# B&R Automation Studio project EFI (part 11)

#### StackMethods.st
```iecst
ACTION StackMethods:

	IF NOT dataHeigh.status.xNewMediaStackEnabled THEN
		EnteringMediaContinuous.Media := dataHeigh.parameters.ContinuousMedia.MediaData;
	END_IF

	ReviewLoadNewMediaMethod;
	ReviewInsertNewMedia;
	ReviewRemoveNewMedia;

	ReviewLoadNewMediaEnergyMethod;
	ReviewInsertNewMediaEnMethod;

	ReviewLoadNewMediaEnergyContMethod;

	dataHeigh.status.Stack.iNewMediaLoadedL1 := Stack_iTotalNewMediaL1;
	dataHeigh.status.Stack.iNewMediaLoadedL2 := Stack_iTotalNewMediaL2;

END_ACTION

ACTION ReviewLoadNewMediaMethod:

	CASE LoadNewMedia_Step OF
		0: // Manage errors and init
			LoadNewMedia_Step := 1;

		1: // start operate
			LoadNewMedia_MethodOperate.Action  := UaMoa_CheckIsCalled;
			LoadNewMedia_MethodOperate.MethodName := 'LoadNewMedia';
			LoadNewMedia_MethodOperate.Execute := TRUE;
			LoadNewMedia_Step := 2;
		2: // check if method called
			LoadNewMedia_MethodOperate();
			IF LoadNewMedia_MethodOperate.Busy THEN
				LoadNewMedia_MethodOperate.Execute := FALSE;
			ELSE
				IF LoadNewMedia_MethodOperate.Done THEN
					LoadNewMedia_ErrorID:= 0;
					IF LoadNewMedia_MethodOperate.IsCalled THEN
						LoadNewMedia_Step := 3; // method is called
					END_IF
					LoadNewMedia_MethodOperate.Execute := TRUE;
				END_IF
				IF LoadNewMedia_MethodOperate.Error THEN
					LoadNewMedia_ErrorID:= DWORD_TO_UDINT(LoadNewMedia_MethodOperate.ErrorID);
					LoadNewMedia_Step := 0;
				END_IF
			END_IF
		3: // execute method code and return value
			ExecuteLoadingNewMedia;
			LoadNewMedia_Result := LoadNewMedia_ReviewResult;
			LoadNewMedia_Step := 4;
		4: // finish operate

			LoadNewMedia_MethodOperate.Action  := UaMoa_Finished;
			LoadNewMedia_MethodOperate.MethodName := 'LoadNewMedia';
			LoadNewMedia_MethodOperate.Execute := TRUE;
			LoadNewMedia_Step := 5;
		5: // finish method
			LoadNewMedia_MethodOperate();
			IF LoadNewMedia_MethodOperate.Busy THEN
				LoadNewMedia_MethodOperate.Execute := FALSE;
			ELSE
				IF LoadNewMedia_MethodOperate.Done THEN
					LoadNewMedia_ErrorID:= 0;
					LoadNewMedia_Step := 1; // method is finished, wait again for call
				END_IF
				IF LoadNewMedia_MethodOperate.Error THEN
					LoadNewMedia_ErrorID:= DWORD_TO_UDINT(LoadNewMedia_MethodOperate.ErrorID);
					LoadNewMedia_Step := 0;
				END_IF
			END_IF
	END_CASE

END_ACTION

ACTION ExecuteLoadingNewMedia:

	LoadNewMedia_ReviewResult := CheckMediaToStack(LoadNewMedia_Media,
												dataHeigh.status.xNewMediaStackEnabled,
												dataHeigh.parameters.xDoubleLine,
												25,
												200, 1400,
												200, 3000,
												Stack_iTotalNewMediaL1 >= THICK_MEDIATRACKING_MAX_MEDIA,
												Stack_iTotalNewMediaL2 >= THICK_MEDIATRACKING_MAX_MEDIA);

	IF LoadNewMedia_ReviewResult <> 0 THEN
		RETURN;
	END_IF

	// TODO: Load the media in the FIFO to manage it
	IF LoadNewMedia_Media.iLine = 1 THEN
		LoadNewMedia_ReviewResult := AssignLastItemInStack(
			ADR(LoadNewMedia_Media),
			ADR(NewMediaStackL1),
			Stack_iTotalNewMediaL1);

	ELSIF LoadNewMedia_Media.iLine = 2 THEN
		LoadNewMedia_ReviewResult := AssignLastItemInStack(
			ADR(LoadNewMedia_Media),
			ADR(NewMediaStackL2),
			Stack_iTotalNewMediaL2);

	END_IF

END_ACTION

ACTION ReviewInsertNewMedia:

	CASE InsertNewMedia_Step OF
		0: // Manage errors and init
			InsertNewMedia_Step := 1;

		1: // start operate
			InsertNewMedia_MethodOperate.Action  := UaMoa_CheckIsCalled;
			InsertNewMedia_MethodOperate.MethodName := 'InsertNewMedia';
			InsertNewMedia_MethodOperate.Execute := TRUE;
			InsertNewMedia_Step := 2;
		2: // check if method called
			InsertNewMedia_MethodOperate();
			IF InsertNewMedia_MethodOperate.Busy THEN
				InsertNewMedia_MethodOperate.Execute := FALSE;
			ELSE
				IF InsertNewMedia_MethodOperate.Done THEN
					InsertNewMedia_ErrorID:= 0;
					IF InsertNewMedia_MethodOperate.IsCalled THEN
						InsertNewMedia_Step := 3; // method is called
					END_IF
					InsertNewMedia_MethodOperate.Execute := TRUE;
				END_IF
				IF InsertNewMedia_MethodOperate.Error THEN
					InsertNewMedia_ErrorID:= DWORD_TO_UDINT(InsertNewMedia_MethodOperate.ErrorID);
					InsertNewMedia_Step := 0;
				END_IF
			END_IF
		3: // execute method code and return value
			ExecuteInsertNewMedia;
			InsertNewMedia_Result := InsertNewMedia_ReviewResult;
			InsertNewMedia_Step := 4;
		4: // finish operate

			InsertNewMedia_MethodOperate.Action  := UaMoa_Finished;
			InsertNewMedia_MethodOperate.MethodName := 'InsertNewMedia';
			InsertNewMedia_MethodOperate.Execute := TRUE;
			InsertNewMedia_Step := 5;
		5: // finish method
			InsertNewMedia_MethodOperate();
			IF InsertNewMedia_MethodOperate.Busy THEN
				InsertNewMedia_MethodOperate.Execute := FALSE;
			ELSE
				IF InsertNewMedia_MethodOperate.Done THEN
					InsertNewMedia_ErrorID:= 0;
					InsertNewMedia_Step := 1; // method is finished, wait again for call
				END_IF
				IF InsertNewMedia_MethodOperate.Error THEN
					InsertNewMedia_ErrorID:= DWORD_TO_UDINT(InsertNewMedia_MethodOperate.ErrorID);
					InsertNewMedia_Step := 0;
				END_IF
			END_IF
	END_CASE

END_ACTION

ACTION ExecuteInsertNewMedia:

	InsertNewMedia_ReviewResult := CheckMediaToStack(InsertNewMedia_Media,
												dataHeigh.status.xNewMediaStackEnabled,
												dataHeigh.parameters.xDoubleLine,
												25,
												200, 1400,
												200, 3000,
												Stack_iTotalNewMediaL1 >= THICK_MEDIATRACKING_MAX_MEDIA,
												Stack_iTotalNewMediaL2 >= THICK_MEDIATRACKING_MAX_MEDIA);

	IF InsertNewMedia_ReviewResult <> 0 THEN
		RETURN;
	END_IF

	// Load the media in the FIFO to manage it.
	// If an error occurs, the error is stored to return it in the method
	IF InsertNewMedia_Media.iLine = 1 THEN
		InsertNewMedia_ReviewResult := InsertItemInStack(
			InsertNewMedia_Id,
			ADR(InsertNewMedia_Media),
			ADR(NewMediaStackL1),
			//InsertNewMedia_Position,
			Stack_iTotalNewMediaL1
		);
	ELSIF InsertNewMedia_Media.iLine = 2 THEN
		InsertNewMedia_ReviewResult := InsertItemInStack(
			InsertNewMedia_Id,
			ADR(InsertNewMedia_Media),
			ADR(NewMediaStackL2),
			//InsertNewMedia_Position,
			Stack_iTotalNewMediaL2
		);
	END_IF

END_ACTION

ACTION ReviewRemoveNewMedia:

	CASE RemoveNewMedia_Step OF
		0: // Manage errors and init
			RemoveNewMedia_Step := 1;

		1: // start operate
			RemoveNewMedia_MethodOperate.Action  := UaMoa_CheckIsCalled;
			RemoveNewMedia_MethodOperate.MethodName := 'RemoveNewMedia';
			RemoveNewMedia_MethodOperate.Execute := TRUE;
			RemoveNewMedia_Step := 2;
		2: // check if method called
			RemoveNewMedia_MethodOperate();
			IF RemoveNewMedia_MethodOperate.Busy THEN
				RemoveNewMedia_MethodOperate.Execute := FALSE;
			ELSE
				IF RemoveNewMedia_MethodOperate.Done THEN
					RemoveNewMedia_ErrorID:= 0;
					IF RemoveNewMedia_MethodOperate.IsCalled THEN
						RemoveNewMedia_Step := 3; // method is called
					END_IF
					RemoveNewMedia_MethodOperate.Execute := TRUE;
				END_IF
				IF RemoveNewMedia_MethodOperate.Error THEN
					RemoveNewMedia_ErrorID:= DWORD_TO_UDINT(RemoveNewMedia_MethodOperate.ErrorID);
					RemoveNewMedia_Step := 0;
				END_IF
			END_IF
		3: // execute method code and return value
			ExecuteRemoveNewMedia;
			RemoveNewMedia_Result := RemoveNewMedia_ReviewResult;
			RemoveNewMedia_Step := 4;
		4: // finish operate

			RemoveNewMedia_MethodOperate.Action  := UaMoa_Finished;
			RemoveNewMedia_MethodOperate.MethodName := 'RemoveNewMedia';
			RemoveNewMedia_MethodOperate.Execute := TRUE;
			RemoveNewMedia_Step := 5;
		5: // finish method
			RemoveNewMedia_MethodOperate();
			IF RemoveNewMedia_MethodOperate.Busy THEN
				RemoveNewMedia_MethodOperate.Execute := FALSE;
			ELSE
				IF RemoveNewMedia_MethodOperate.Done THEN
					RemoveNewMedia_ErrorID:= 0;
					RemoveNewMedia_Step := 1; // method is finished, wait again for call
				END_IF
				IF RemoveNewMedia_MethodOperate.Error THEN
					RemoveNewMedia_ErrorID:= DWORD_TO_UDINT(RemoveNewMedia_MethodOperate.ErrorID);
					RemoveNewMedia_Step := 0;
				END_IF
			END_IF
	END_CASE

END_ACTION

ACTION ExecuteRemoveNewMedia:

	RemoveNewMedia_ReviewResult := CheckLineToStack(RemoveNewMedia_Line,
												dataHeigh.status.xNewMediaStackEnabled,
												dataHeigh.parameters.xDoubleLine);

	IF RemoveNewMedia_ReviewResult <> 0 THEN
		RETURN;
	END_IF

	// TODO: Load the media in the FIFO to manage it
	IF RemoveNewMedia_Line = 1 THEN
		RemoveNewMedia_ReviewResult := RemoveItemInStack(RemoveNewMedia_Id, ADR(NewMediaStackL1), Stack_iTotalNewMediaL1);
	ELSIF RemoveNewMedia_Line = 2 THEN
		RemoveNewMedia_ReviewResult := RemoveItemInStack(RemoveNewMedia_Id, ADR(NewMediaStackL2), Stack_iTotalNewMediaL2);
	END_IF

END_ACTION

ACTION ReviewLoadNewMediaEnergyMethod:

	CASE LoadNewMediaEnergy_Step OF
		0: // Manage errors and init
			LoadNewMediaEnergy_Step := 1;

		1: // start operate
			LoadNewMediaEnergy_MethodOperate.Action  := UaMoa_CheckIsCalled;
			LoadNewMediaEnergy_MethodOperate.MethodName := 'LoadNewMediaEnergy';
			LoadNewMediaEnergy_MethodOperate.Execute := TRUE;
			LoadNewMediaEnergy_Step := 2;
		2: // check if method called
			LoadNewMediaEnergy_MethodOperate();
			IF LoadNewMediaEnergy_MethodOperate.Busy THEN
				LoadNewMediaEnergy_MethodOperate.Execute := FALSE;
			ELSE
				IF LoadNewMediaEnergy_MethodOperate.Done THEN
					LoadNewMediaEnergy_ErrorID:= 0;
					IF LoadNewMediaEnergy_MethodOperate.IsCalled THEN
						LoadNewMediaEnergy_Step := 3; // method is called
					END_IF
					LoadNewMediaEnergy_MethodOperate.Execute := TRUE;
				END_IF
				IF LoadNewMediaEnergy_MethodOperate.Error THEN
					LoadNewMediaEnergy_ErrorID:= DWORD_TO_UDINT(LoadNewMediaEnergy_MethodOperate.ErrorID);
					LoadNewMediaEnergy_Step := 0;
				END_IF
			END_IF
		3: // execute method code and return value
			ExecuteLoadingNewMediaEnergy;
			LoadNewMediaEnergy_Result := LoadNewMediaEnergy_ReviewResult;
			LoadNewMediaEnergy_Step := 4;
		4: // finish operate

			LoadNewMediaEnergy_MethodOperate.Action  := UaMoa_Finished;
			LoadNewMediaEnergy_MethodOperate.MethodName := 'LoadNewMediaEnergy';
			LoadNewMediaEnergy_MethodOperate.Execute := TRUE;
			LoadNewMediaEnergy_Step := 5;
		5: // finish method
			LoadNewMediaEnergy_MethodOperate();
			IF LoadNewMediaEnergy_MethodOperate.Busy THEN
				LoadNewMediaEnergy_MethodOperate.Execute := FALSE;
			ELSE
				IF LoadNewMediaEnergy_MethodOperate.Done THEN
					LoadNewMediaEnergy_ErrorID:= 0;
					LoadNewMediaEnergy_Step := 1; // method is finished, wait again for call
				END_IF
				IF LoadNewMediaEnergy_MethodOperate.Error THEN
					LoadNewMediaEnergy_ErrorID:= DWORD_TO_UDINT(LoadNewMediaEnergy_MethodOperate.ErrorID);
					LoadNewMediaEnergy_Step := 0;
				END_IF
			END_IF
	END_CASE

END_ACTION

ACTION ExecuteLoadingNewMediaEnergy:

	LoadNewMediaEnergy_ReviewResult := CheckMediaToStack(LoadNewMediaEnergy_Media.MediaData,
												dataHeigh.parameters.Dry.xDryStack,
												dataHeigh.parameters.xDoubleLine,
												25,
												200, 1400,
												200, 3000,
												Stack_iTotalNewMediaL1 >= THICK_MEDIATRACKING_MAX_MEDIA,
												Stack_iTotalNewMediaL2 >= THICK_MEDIATRACKING_MAX_MEDIA);

	IF LoadNewMediaEnergy_ReviewResult <> 0 THEN
		RETURN;
	END_IF

	// TODO: Check the final dimensions of the media

	// Load the media in the FIFO to manage it
	IF LoadNewMediaEnergy_Media.MediaData.iLine = 1 THEN
		LoadNewMediaEnergy_ReviewResult := AssignLastItemEnergyInStack(
			ADR(LoadNewMediaEnergy_Media.MediaData),
			ADR(LoadNewMediaEnergy_Media.Energy),
			ADR(NewMediaStackL1),
			ADR(MediaEnergyRackL1),
			Stack_iTotalNewMediaL1,
			EnergyRack_iIndexL1);

	ELSIF LoadNewMediaEnergy_Media.MediaData.iLine = 2 THEN
		LoadNewMediaEnergy_ReviewResult := AssignLastItemEnergyInStack(
			ADR(LoadNewMediaEnergy_Media.MediaData),
			ADR(LoadNewMediaEnergy_Media.Energy),
			ADR(NewMediaStackL2),
			ADR(MediaEnergyRackL2),
			Stack_iTotalNewMediaL2,
			EnergyRack_iIndexL2);

	END_IF

END_ACTION

ACTION ReviewInsertNewMediaEnMethod:

	CASE InsertNewMediaEn_Step OF
		0: // Manage errors and init
			InsertNewMediaEn_Step := 1;

		1: // start operate
			InsertNewMediaEn_MethodOperate.Action  := UaMoa_CheckIsCalled;
			InsertNewMediaEn_MethodOperate.MethodName := 'InsertNewMediaEnergy';
			InsertNewMediaEn_MethodOperate.Execute := TRUE;
			InsertNewMediaEn_Step := 2;
		2: // check if method called
			InsertNewMediaEn_MethodOperate();
			IF InsertNewMediaEn_MethodOperate.Busy THEN
				InsertNewMediaEn_MethodOperate.Execute := FALSE;
			ELSE
				IF InsertNewMediaEn_MethodOperate.Done THEN
					InsertNewMediaEn_ErrorID:= 0;
					IF InsertNewMediaEn_MethodOperate.IsCalled THEN
						InsertNewMediaEn_Step := 3; // method is called
					END_IF
					InsertNewMediaEn_MethodOperate.Execute := TRUE;
				END_IF
				IF InsertNewMediaEn_MethodOperate.Error THEN
					InsertNewMediaEn_ErrorID:= DWORD_TO_UDINT(InsertNewMediaEn_MethodOperate.ErrorID);
					InsertNewMediaEn_Step := 0;
				END_IF
			END_IF
		3: // execute method code and return value
			ExecuteInsertNewMediaEn;
			InsertNewMediaEn_Result := InsertNewMediaEn_ReviewResult;
			InsertNewMediaEn_Step := 4;
		4: // finish operate

			InsertNewMediaEn_MethodOperate.Action  := UaMoa_Finished;
			InsertNewMediaEn_MethodOperate.MethodName := 'InsertNewMediaEnergy';
			InsertNewMediaEn_MethodOperate.Execute := TRUE;
			InsertNewMediaEn_Step := 5;
		5: // finish method
			InsertNewMediaEn_MethodOperate();
			IF InsertNewMediaEn_MethodOperate.Busy THEN
				InsertNewMediaEn_MethodOperate.Execute := FALSE;
			ELSE
				IF InsertNewMediaEn_MethodOperate.Done THEN
					InsertNewMediaEn_ErrorID:= 0;
					InsertNewMediaEn_Step := 1; // method is finished, wait again for call
				END_IF
				IF InsertNewMediaEn_MethodOperate.Error THEN
					InsertNewMediaEn_ErrorID:= DWORD_TO_UDINT(InsertNewMediaEn_MethodOperate.ErrorID);
					InsertNewMediaEn_Step := 0;
				END_IF
			END_IF
	END_CASE

END_ACTION

ACTION ExecuteInsertNewMediaEn:

	InsertNewMediaEn_ReviewResult := CheckMediaToStack(InsertNewMediaEn_Media.MediaData,
													dataHeigh.parameters.Dry.xDryStack,
													dataHeigh.parameters.xDoubleLine,
													25,
													200, 1400,
													200, 3000,
													Stack_iTotalNewMediaL1 >= THICK_MEDIATRACKING_MAX_MEDIA,
													Stack_iTotalNewMediaL2 >= THICK_MEDIATRACKING_MAX_MEDIA);

	IF InsertNewMediaEn_ReviewResult <> 0 THEN
		RETURN;
	END_IF

	// TODO: Load the media in the FIFO to manage it
	IF InsertNewMediaEn_Media.MediaData.iLine = 1 THEN
		// Addign new media to after a defined position
		InsertNewMediaEn_ReviewResult := InsertItemEnergyInStack(
			InsertNewMediaEn_Id,
			ADR(InsertNewMediaEn_Media.MediaData),
			ADR(InsertNewMediaEn_Media.Energy),
			ADR(NewMediaStackL1),
			ADR(MediaEnergyRackL1),
			Stack_iTotalNewMediaL1,
			EnergyRack_iIndexL1);

	ELSIF InsertNewMediaEn_Media.MediaData.iLine = 2 THEN
		// Addign new media to after a defined position
		InsertNewMediaEn_ReviewResult := InsertItemEnergyInStack(
			InsertNewMediaEn_Id,
			ADR(InsertNewMediaEn_Media.MediaData),
			ADR(InsertNewMediaEn_Media.Energy),
			ADR(NewMediaStackL2),
			ADR(MediaEnergyRackL2),
			Stack_iTotalNewMediaL2,
			EnergyRack_iIndexL2);

	END_IF

END_ACTION

ACTION ReviewLoadNewMediaEnergyContMethod:

	CASE LoadNewMediaEnergyCont_Step OF
		0: // Manage errors and init
			LoadNewMediaEnergyCont_Step := 1;

		1: // start operate
			LoadNewMediaEnergyCont_MethodOp.Action  := UaMoa_CheckIsCalled;
			LoadNewMediaEnergyCont_MethodOp.MethodName := 'LoadNewMediaEnergyCont';
			LoadNewMediaEnergyCont_MethodOp.Execute := TRUE;
			LoadNewMediaEnergyCont_Step := 2;
		2: // check if method called
			LoadNewMediaEnergyCont_MethodOp();
			IF LoadNewMediaEnergyCont_MethodOp.Busy THEN
				LoadNewMediaEnergyCont_MethodOp.Execute := FALSE;
			ELSE
				IF LoadNewMediaEnergyCont_MethodOp.Done THEN
					LoadNewMediaEnergyCont_ErrorID:= 0;
					IF LoadNewMediaEnergyCont_MethodOp.IsCalled THEN
						LoadNewMediaEnergyCont_Step := 3; // method is called
					END_IF
					LoadNewMediaEnergyCont_MethodOp.Execute := TRUE;
				END_IF
				IF LoadNewMediaEnergyCont_MethodOp.Error THEN
					LoadNewMediaEnergyCont_ErrorID:= DWORD_TO_UDINT(LoadNewMediaEnergyCont_MethodOp.ErrorID);
					LoadNewMediaEnergyCont_Step := 0;
				END_IF
			END_IF
		3: // execute method code and return value
			ExecuteLoadingNewMediaEnergyCont;
			LoadNewMediaEnergyCont_Result := LoadNewMediaEnergyCont_ReviewRes;
			LoadNewMediaEnergyCont_Step := 4;
		4: // finish operate

			LoadNewMediaEnergyCont_MethodOp.Action  := UaMoa_Finished;
			LoadNewMediaEnergyCont_MethodOp.MethodName := 'LoadNewMediaEnergyCont';
			LoadNewMediaEnergyCont_MethodOp.Execute := TRUE;
			LoadNewMediaEnergyCont_Step := 5;
		5: // finish method
			LoadNewMediaEnergyCont_MethodOp();
			IF LoadNewMediaEnergyCont_MethodOp.Busy THEN
				LoadNewMediaEnergyCont_MethodOp.Execute := FALSE;
			ELSE
				IF LoadNewMediaEnergyCont_MethodOp.Done THEN
					LoadNewMediaEnergyCont_ErrorID:= 0;
					LoadNewMediaEnergyCont_Step := 1; // method is finished, wait again for call
				END_IF
				IF LoadNewMediaEnergyCont_MethodOp.Error THEN
					LoadNewMediaEnergyCont_ErrorID:= DWORD_TO_UDINT(LoadNewMediaEnergyCont_MethodOp.ErrorID);
					LoadNewMediaEnergyCont_Step := 0;
				END_IF
			END_IF
	END_CASE

END_ACTION

ACTION ExecuteLoadingNewMediaEnergyCont:

	LoadNewMediaEnergyCont_ReviewRes := CheckMediaToStack(LoadNewMediaEnergyCont_Media.MediaData,
													TRUE,
													dataHeigh.parameters.xDoubleLine,
													25,
													200, 1400,
													200, 3000,
													Stack_iTotalNewMediaL1 >= THICK_MEDIATRACKING_MAX_MEDIA,
													Stack_iTotalNewMediaL2 >= THICK_MEDIATRACKING_MAX_MEDIA);

	IF LoadNewMediaEnergyCont_ReviewRes <> 0 THEN
		RETURN;
	END_IF

	// TODO: Check the final dimensions of the media
	dataHeigh.parameters.ContinuousMedia := LoadNewMediaEnergyCont_Media;
	IF dataHeigh.parameters.pExtContMedia > 0 THEN
		ExternalMediaConfig ACCESS dataHeigh.parameters.pExtContMedia;
		ExternalMediaConfig := dataHeigh.parameters.ContinuousMedia.MediaData;
	END_IF

END_ACTION
```

### Program Logical/ExtPack/_Media/ThicknessCtrl/ThicknessCtrl_v2/ThickReadEnergy (IEC) - Cyclic code

#### ThickReadEnergy.var
```iecst
(********************************************************************
 * COPYRIGHT -- Bernecker + Rainer
 ********************************************************************
 * Program: FileHandling
 * File: FileHandling.var
 * Author: Bernecker + Rainer
 * Created: April 16, 2009
 ********************************************************************
 * Local variables of program FileHandling
 ********************************************************************)
VAR
	Handling : FileHandling_typ := (0); (*Handlingdata for this fileio example*)
	Select : USINT; (*variable to select the file-device*)
	Error : UINT; (*return value from FileIoGetSysError()*)
END_VAR
```

### Program Logical/ExtPack/_Media/ThicknessCtrl/ThicknessCtrlSim/ThicknessCtrlSim_v1/ThicknessCtrlSim (IEC)

#### ThicknessCtrlSim.st
```iecst
PROGRAM _INIT

END_PROGRAM

PROGRAM _CYCLIC

	// Moved from init to cyclic. This cannot be in init because sim is executed before ThicknessCtrl and the assignement is done in ThicknessCtrl INIT
	xMediaTracking ACCESS gThicknessCtrl.Internal.pMediaTracking;
	iDistanceWorkEmptyBelt ACCESS gThicknessCtrl.Internal.pDistanceWorkEmptyBelt;

	IF NOT gSimThickCtrl.Orders.NotActivateMediaInPos THEN
		gThicknessCtrl.Inputs.CheckMedia[1].xCheckFail := xMediaTracking[gThicknessCtrl.parameters.CheckMedia[1].CheckPosition] > 0;
		gThicknessCtrl.Inputs.CheckMedia[2].xCheckFail := xMediaTracking[gThicknessCtrl.parameters.CheckMedia[2].CheckPosition] > 0;
	ELSE
		gThicknessCtrl.Inputs.CheckMedia[1].xCheckFail := FALSE;
		gThicknessCtrl.Inputs.CheckMedia[2].xCheckFail := FALSE;
	END_IF

	// Related to NOZOMITWO-2388
	IF gSimThickCtrl.Commands.xEmptyMediaTracking THEN
		FOR iIndexMediaTrack := 0 TO iMAXTRACKINGARRAY DO
			xMediaTracking[iIndexMediaTrack] := 0;
			iDistanceWorkEmptyBelt := 0;
		END_FOR
		gSimThickCtrl.Commands.xEmptyMediaTracking := FALSE;
	END_IF

END_PROGRAM

PROGRAM _EXIT
	(* Insert code here *)

END_PROGRAM
```

### ThicknessCtrlSim.typ
```iecst
TYPE
	SimThickCtrlOrders_typ : 	STRUCT
		NotActivateMediaInPos : BOOL; (*Do not activate the right behavior of activating the signal when media is detected*)
	END_STRUCT;
	SimThickCtrlCommands_typ : 	STRUCT
		xEmptyMediaTracking : BOOL;
	END_STRUCT;
	SimThickCtrlParams_typ : 	STRUCT
		New_Member : BOOL;
	END_STRUCT;
	SimThickCtrl_typ : 	STRUCT
		Commands : SimThickCtrlCommands_typ;
		Orders : SimThickCtrlOrders_typ;
		Parameters : SimThickCtrlParams_typ;
	END_STRUCT;
END_TYPE
```

### Program Logical/ExtPack/_Media/nSensorCtrl/nSensorCtrl_v2/nSensorCtrl (IEC)

#### nSensorCtrl.st - Init, cyclic, exit code
```iecst
PROGRAM _INIT
	FOR iIndexHistory:=0  TO iHistoryLines DO
		StateHistory[iIndexHistory]:=STP_NOT_USED;
	END_FOR;
END_PROGRAM

PROGRAM _CYCLIC

	//////////////////////////////
	////// ASIGN LOCAL VARS //////
	//////////////////////////////

	//Main data assignation
	data 	ACCESS ADR (gPhotoCells);
	// Assign Stepper Motor reference
	Stepper 	ACCESS ADR (gAxis[data.parameters.IndexDriveMaster]);
	StepperGear ACCESS ADR (gAxis[data.parameters.IndexDriveSecondary]);
	Icla 		ACCESS ADR (gIcla[data.parameters.IndexIcla]);

	// Assigning status.xInstalled considering dynamic enable
	IF data.parameters.xInstall THEN
		IF data.parameters.xAllowDynamicEnable THEN
			data.status.xInstalled:= data.parameters.xEnable;
		ELSE
			data.status.xInstalled:= TRUE;
		END_IF
	ELSE
		data.status.xInstalled:= FALSE;
	END_IF

	//To reset status when motor type is modified. Not likely to occur in field. Discovered while simulating several platforms in a row.
	xMotorChanged := PreviousMotorType <> data.parameters.MotorType;
	PreviousMotorType := data.parameters.MotorType;

	IF NOT data.status.xInstalled OR xMotorChanged THEN

		// Reset alarms 3L
		data.Alarms:=stnSensorsAlarmsReseted ;
		data.AlSummary := stnSensorsAlarmSummaryReseted;
		data.AlSummary.xAlarmSound:=FALSE;

		data.status.xReferenced:=FALSE;
		data.status.xSensorValidAlignPos := FALSE;
		data.status.xLowPieceDetect := FALSE;

		RETURN;
	END_IF

	data.parameters.iSensorQuantity := LIMIT(2, data.parameters.iSensorQuantity, MAX_LAST_NSENSOR);
	data.parameters.iSensorToReference := LIMIT(1, data.parameters.iSensorToReference, MAX_LAST_NSENSOR);

	/////////////////////////
	// MOTOR PARAMETERS /////
	/////////////////////////

	DataToMotors;

	// 3 Photocells position to machine ctrl
	// Photocells are not moving when when photocells is detecting tile, In auto it goes to referenced position
	IF data.commands.AutoMode.xBypass AND gPhotoCells.parameters.xEnableMountedAlrByPass THEN
		rSensorPositionDesired:= data.parameters.rSensorMechPositionByPass;
	ELSE
		IF data.status.xSensorsPositionedRelativeToBar THEN
			rSensorPositionDesired:= data.status.rOffsetToApplyToBarsPosition;
		ELSE
			rSensorPositionDesired:= data.parameters.rMediaThickness + data.parSw.rMechOffset + data.parameters.rOffsetPosition;
		END_IF

	END_IF

	DataFromMotors;

	xAllSensorInactive := TRUE;
	xAllSensorActive := TRUE;
	FOR iIndexSensor:=1 TO data.parameters.iSensorQuantity DO
		IF data.Inputs.Signals.xPhotoCells[iIndexSensor] THEN
			xAllSensorInactive:= FALSE;
		ELSE
			xAllSensorActive:= FALSE;
		END_IF

		IF data.parameters.Sensors[iIndexSensor].xEnabled THEN
			IF iIndexSensor<>1 AND iIndexSensor<>data.parameters.iSensorQuantity THEN
				IF data.status.xSensorsPositionedRelativeToBar THEN
					data.parameters.Sensors[iIndexSensor].xMoveBarsUp := iIndexSensor>=data.status.iSensorToApplyOffset;
				ELSE
					data.parameters.Sensors[iIndexSensor].xMoveBarsUp := TRUE;
				END_IF
			END_IF
		ELSE
			data.parameters.Sensors[iIndexSensor].xMoveBarsUp := FALSE;
			data.parameters.Sensors[iIndexSensor].xMountedMedia := FALSE;
		END_IF

		//Always, for all machine models, the only photocell enabled to active mounted media alarm is the last one (highest positioned)
		IF iIndexSensor=data.parameters.iSensorQuantity THEN
			data.parameters.Sensors[iIndexSensor].xMountedMedia := TRUE;
		END_IF

		//Writting distance to belt surface for each sensor
		data.parameters.Sensors[iIndexSensor].rDistanceToBase := data.parameters.Sensors[iIndexSensor].rDistanceRelativeToFirstSensor + data.status.rPositionMotor;

		//NOZOMITWO-2066: Checking that all sensors positioned above one selected to reject media, are defined to reject media too.
		IF iIndexSensor<data.parameters.iSensorQuantity THEN
			IF data.parSw.Sensors[iIndexSensor].xToRejectMedia THEN
				data.parSw.Sensors[iIndexSensor+1].xToRejectMedia := TRUE;
			END_IF
		END_IF

	END_FOR

	//Defining sensors behaviour
	IF data.parameters.xSensorsPosHybridBehaviour THEN
		xSensorsPositionedRelativeToBar := FALSE;
		data.status.xSensorsPositionedRelativeToBar := FALSE;

		FOR iIndexSensorToPositionBelowBars:=2 TO (data.parameters.iSensorQuantity-1) DO
			rOffsetPositionCalc := data.parameters.rMediaThickness + data.parameters.rMarginPrint - data.parameters.Sensors[iIndexSensorToPositionBelowBars].rDistanceRelativeToFirstSensor - data.parameters.rOffsetRelToBar;
			IF (rOffsetPositionCalc<=data.parameters.rMediaThickness-0.5) THEN
				IF (rOffsetPositionCalc>=0.5) THEN
					//Save index of the sensor positioned below bars
					data.status.iSensorToApplyOffset:=iIndexSensorToPositionBelowBars;

					//To set first photocell position
					rOffsetPosition:=rOffsetPositionCalc;

					//Photocell A must be positioned above the belt
					xSensorsPositionedRelativeToBar := TRUE;
					EXIT;
				END_IF
			END_IF
		END_FOR
		data.status.xSensorsPositionedRelativeToBar := xSensorsPositionedRelativeToBar;
	ELSE
		data.status.xSensorsPositionedRelativeToBar := FALSE;
	END_IF

	data.status.rOffsetToApplyToBarsPosition := rOffsetPosition;

	data.status.xAllPhotoInactive:= xAllSensorInactive;
	data.status.xTrustPhotocellASignal := data.status.rPositionMotor>0.5; //Sensor light beam diameter is 1mm

	///////////////////////////////////////////////
	////// nSensorCtrl MachineState  //////////////
	///////////////////////////////////////////////
	MachineState;

	/////////////////////////
	////// ALARMS ///////////
	/////////////////////////
	AlarmsSummary;

	///////////////////////
	//Alarm Sound
	AlarmSounds;

	///////////////////////////
	// Mounted media management. ThicknessCtrl MUST be executed in the slow cycle before this program
	IF data.status.xMountedMediaDetected AND NOT data._Internal.xMountedMediaTreated THEN
		data._Internal.xMountedMediaTreated := TRUE;
	END_IF
	IF NOT data.status.xMountedMediaDetected THEN
		data._Internal.xMountedMediaTreated := FALSE;
	END_IF

	///////////////////////////
	// Media To Reject management. ThicknessCtrl MUST be executed in the slow cycle before this program
	IF data.status.xMediaToRejectDetected AND NOT data._Internal.xMediaToRejectTreated THEN
		data._Internal.xMediaToRejectTreated := TRUE;
	END_IF
	IF NOT data.status.xMediaToRejectDetected THEN
		data._Internal.xMediaToRejectTreated := FALSE;
	END_IF

	data.status.rOffsetToReject := data.parameters.Sensors[iWarpMediaSensor].rDistanceRelativeToFirstSensor;
	data.status.rOffsetToMounted := data.parameters.Sensors[data.parameters.iSensorQuantity].rDistanceRelativeToFirstSensor;

	xPhotoInputsPrev := data.Inputs.Signals.xPhotoCells;

	//Resetting commands coming from sw
	data.commandsSw := ResetCommandsSw;

END_PROGRAM
```

#### AlarmsSummary.st - nSensors alarms summary
```iecst
ACTION AlarmsSummary:

	//////////////////////////
	////// RESET ALARMS //////
	//////////////////////////
	// Pending do commands gdata.commands.xReset
	IF data.commands.xErrorRst THEN
		data.Alarms := stnSensorsAlarmsReseted;
		data.AlSummary := stnSensorsAlarmSummaryReseted;
	END_IF

	//Invalid positions
	data.Alarms.xAlrInvalidAlignmentPosition:= NOT data.status.xSensorValidAlignPos AND (data.parameters.AlignmentProcess = STP_ALIGNMENT_REQUIRED);

	//MaxPositionReached just while searching alignement
	iStateToCheckPosition.0 := data.status.iSystemState = STP_SEARCH_ALIGNMENT_POS_STEP_1;
	iStateToCheckPosition.1 := data.status.iSystemState = STP_SEARCH_ALIGNMENT_POS_STEP_2;
	iStateToCheckPosition.2 := data.status.iSystemState = STP_SEARCH_ALIGNMENT_POS_STEP_3;
	iStateToCheckPosition.3 := data.status.iSystemState = STP_RUNING AND data.status.xReferenced;
	iStateToCheckPosition.4 := data.status.iSystemState = STP_STANDSTILL;

	IF iStateToCheckPosition > 0 THEN
		iLastStateToCheckPosition := iStateToCheckPosition;

		IF ((rPositionMotorMm > data.parameters.rSensorMechPositionMax) OR (rPositionMotorMm < data.parameters.rSensorMechPositionMin)) THEN
			data.Alarms.xPositionOutOfRange := TRUE;
		END_IF
	END_IF

	IF NOT data.Alarms.xAlrInvalidAlignmentPosition THEN
		//Operational photocells must be evaluated too: detecting ones and first enabled for mounted alarm
		FOR iIndexSensor:=1 TO data.parameters.iSensorQuantity DO
			IF data.status.xPhotoCellsNotAligned[iIndexSensor] THEN
				IF ((NOT data.parameters.Sensors[iIndexSensor].xMountedMedia) OR (NOT data.parameters.Sensors[iIndexSensor-1].xMountedMedia)) THEN
					data.Alarms.xAlrCriticalPhotocellNotAligned:= TRUE;
					data.Alarms.xPhotoCellsNotAlignedWarning[iIndexSensor]:= FALSE;
					data.Alarms.xPhotoCellsNotAlignedError[iIndexSensor]:= TRUE;
				ELSE
					data.Alarms.xPhotoCellsNotAlignedWarning[iIndexSensor]:= TRUE;
					data.Alarms.xPhotoCellsNotAlignedError[iIndexSensor]:= FALSE;
				END_IF
			END_IF
		END_FOR
	END_IF

	//Alarm Not referenced
	data.Alarms.xNotReferenced:= NOT data.status.xReferenced;

	// Incoherence Photocells system
	data.status.xSensorsSeparatedInProcessDir := data.parameters.rDistanceBetweenSensors > 0;

	IF data.commands.xCheckMounted THEN
		IF data.status.xSensorsSeparatedInProcessDir THEN
			IncoherenceSensor := 0;
			FOR iIndexSensor:=2 TO data.parameters.iSensorQuantity DO
				IF NOT data.Inputs.Signals.xPhotoCells[iIndexSensor-1] AND data.Inputs.Signals.xPhotoCells[iIndexSensor] AND NOT xPhotoInputsPrev[iIndexSensor] THEN
					data.Alarms.xPhotoCellsDetectionIncoherence[iIndexSensor] := TRUE;
					//These alarms are not considered in alarm sound action. Is just a warning and this avoid to make printer sound very often.
					//To leave it this way till full tested in field
				END_IF
			END_FOR

		ELSE
			IncoherenceSensor.0 := NOT data.Inputs.Signals.xPhotoCells[1] AND data.Inputs.Signals.xPhotoCells[2];
			IncoherenceSensor.1 := NOT data.Inputs.Signals.xPhotoCells[2] AND data.Inputs.Signals.xPhotoCells[3];
			IncoherenceSensor.2 := NOT data.Inputs.Signals.xPhotoCells[3] AND data.Inputs.Signals.xPhotoCells[4];
			IncoherenceSensor.3 := NOT data.Inputs.Signals.xPhotoCells[4] AND data.Inputs.Signals.xPhotoCells[5];
			IncoherenceSensor.4 := NOT data.Inputs.Signals.xPhotoCells[5] AND data.Inputs.Signals.xPhotoCells[6];

			TON_DelayIncoherrPhotocell.IN:= IncoherenceSensor>0 AND data.commands.AutoMode.xProdORLab;
			TON_DelayIncoherrPhotocell.PT:= T#500ms;
			TON_DelayIncoherrPhotocell();

			IF TON_DelayIncoherrPhotocell.Q THEN
				data.Alarms.xIncoherPhotocellSystem:= TRUE;
			END_IF
		END_IF
	END_IF

	// Not comms
	CASE data.parameters.MotorType OF
		STP_STEPPER:
			data.Alarms.xComsMotorError:= (NOT data.status.xBackModuleOk OR NOT data.status.xFrontModuleOk OR Stepper.Status.ErrorID=29365);

		STP_ICLA:
			data.Alarms.xComsMotorError:= Icla.Status.Error.Communication;
	END_CASE

	// Motor Error (Stepper or StepperGear)
	CASE data.parameters.MotorType OF
		STP_STEPPER:
			data.Alarms.xMotorError :=	data.status.xMotorError;

		STP_ICLA:
			data.Alarms.xMotorError := Icla.Status.Error.ErrorNumber<>0;
			data.Alarms.xControllerNotReady := Icla.Status.iDriveStatus = ICLAST_SWITCH_ON_DISABLED AND data.Inputs.Signals.xSafetyEnable AND NOT data.commands.Mode.xZero;
	END_CASE

	//Warp media
	iWarpMediaSensor := data.parameters.iSensorQuantity-1;
	xWarpSensorActive := data.Inputs.Signals.xPhotoCells[iWarpMediaSensor];

	IF data.commands.xCheckMounted AND EDGEPOS(xWarpSensorActive) THEN
		IF NOT xWarpMediaPresent THEN
			iCounterWarpMedia := iCounterWarpMedia+1;
			xWarpMediaPresent := TRUE;
		END_IF

	ELSIF NOT xWarpSensorActive THEN
		xWarpMediaPresent := FALSE;
	END_IF

	IF (iCounterWarpMedia=iMaxWarpMedia) THEN data.Alarms.xAlrWarpMedia:=TRUE; END_IF

	IF NOT data.commands.LineStatusSummary.xPrinting THEN iCounterWarpMedia:=0; END_IF

	//Continuous Reading PD Phcell
	IF data.parameters.MotorType = STP_STEPPER THEN
		TON_ContinuousActPDPhcell.IN := data.Inputs.Signals.xPhotoCells[1] AND data.commands.AutoMode.xProdORLab AND NOT data.commands.AutoMode.xPause;
		TON_ContinuousActPDPhcell.PT := T#30s;
		TON_ContinuousActPDPhcell();

		IF TON_ContinuousActPDPhcell.Q THEN
			data.Alarms.xContinuousActPDPhcell := TRUE;
		END_IF
	END_IF

	//////////////////////////
	////// ALARMS SUMMARY////
	/////////////////////////

	//Stop
	iReasonStop.0 := data.Alarms.xMotorError;
	iReasonStop.1 := data.Alarms.xComsMotorError;
	iReasonStop.2 := data.Alarms.xNotReferenced;
	iReasonStop.3 := data.Alarms.xIncoherPhotocellSystem;
	iReasonStop.4 := data.Alarms.xAlrInvalidAlignmentPosition;
	iReasonStop.5 := data.Alarms.xAlrCriticalPhotocellNotAligned;

	data.AlSummary.xAlarmStop := iReasonStop > 0;
	IF EDGEPOS(data.AlSummary.xAlarmStop) THEN
		data.AlSummary.iReasonStop[0] := iReasonStop;
		LogStopAlarm;
	ELSIF EDGEPOS(NOT data.commands.AutoMode.xStop AND NOT data.AlSummary.xAlarmStop) THEN
		data.AlSummary.iReasonStop[0] := 0;
	END_IF

	//Critical
	iReasonCritical.0 := data.Alarms.xPositionOutOfRange;

	data.AlSummary.xAlarmCritical := iReasonCritical > 0;
	IF EDGEPOS(data.AlSummary.xAlarmCritical) THEN
		data.AlSummary.iReasonCritical := iReasonCritical;
		LogCriticalAlarm;
	ELSIF EDGEPOS(data.commands.Mode.xAuto AND NOT data.AlSummary.xAlarmCritical) THEN
		data.AlSummary.iReasonCritical := 0;
	END_IF

	// It is just used for drive alarms
	iAnyAlarm.0 := data.Alarms.xMotorError;
	iAnyAlarm.1 := data.Alarms.xComsMotorError;
	iAnyAlarm.2 := data.Alarms.xPositionOutOfRange AND data.commands.Mode.xAuto;

	data.AlSummary.xAnyAlarm:= 	iAnyAlarm > 0;

	//Warning
	// It is just used for drive alarms
	iAnyWarning.0 := data.status.xReferencing;
	iAnyWarning.1 := data.Alarms.xNotReferenced;
	iAnyWarning.2 := data.Alarms.xAlrWarpMedia;
	data.AlSummary.xAnyWarning:= iAnyWarning > 0;

	IF EDGEPOS(data.AlSummary.xAnyWarning) THEN
		data.AlSummary.iReasonWarning := iAnyWarning;
		LogWarningAlarm;
	ELSIF EDGEPOS(NOT data.AlSummary.xAnyWarning) THEN
		data.AlSummary.iReasonWarning := 0;
	END_IF

END_ACTION
```

#### AlarmSounds.st
```iecst
ACTION AlarmSounds:

	ars_MotorError.xAlarm:= data.Alarms.xMotorError;
	ars_MotorError.xSilence:= data.commands.xMute;
	ars_MotorError();

	ars_ComsMotorError.xAlarm:= data.Alarms.xComsMotorError;
	ars_ComsMotorError.xSilence:= data.commands.xMute;
	ars_ComsMotorError();

	ars_NotReferenced.xAlarm:= data.Alarms.xNotReferenced;
	ars_NotReferenced.xSilence:= data.commands.xMute;
	ars_NotReferenced();

	ars_IncoherPhotocellSystem.xAlarm:= data.Alarms.xIncoherPhotocellSystem;
	ars_IncoherPhotocellSystem.xSilence:= data.commands.xMute;
	ars_IncoherPhotocellSystem();

	ars_InvalidAlignmentPosition.xAlarm:= data.Alarms.xAlrInvalidAlignmentPosition;
	ars_InvalidAlignmentPosition.xSilence:= data.commands.xMute;
	ars_InvalidAlignmentPosition();

	ars_CriticalPhotocellNotAligned.xAlarm:= data.Alarms.xAlrCriticalPhotocellNotAligned;
	ars_CriticalPhotocellNotAligned.xSilence:= data.commands.xMute;
	ars_CriticalPhotocellNotAligned();

	arsContinuousActPDPhcell.xAlarm:= data.Alarms.xContinuousActPDPhcell;
	arsContinuousActPDPhcell.xSilence:= data.commands.xMute;
	arsContinuousActPDPhcell();

	data.AlSummary.xAlarmSound:= 	ars_MotorError.xAlarmSound OR
									ars_ComsMotorError.xAlarmSound OR
									ars_NotReferenced.xAlarmSound OR
									ars_IncoherPhotocellSystem.xAlarmSound OR
									ars_InvalidAlignmentPosition.xAlarmSound OR
									ars_CriticalPhotocellNotAligned.xAlarmSound OR
									arsContinuousActPDPhcell.xAlarmSound OR
									(xAnyManualOrder AND gPLC.xBlk_200ms);

END_ACTION
```

- PhotoCellStates.graphml - Photocell states ctrl (not shown)

### 3PhotoSens Docu.txt - Block package document
```
#################################################################################
#################################################################################
#																				#
#			GENERAL USE OF 3 PHOTO SENSOR PACKAGE								#
#																				#
# 	To use this 3 Photo Sens unit, some general variables are needed:			#
#																				#
# 		· data 							as nSensors_Generic		#
#		· gAxis	(to Control Master Stepper)		as AxisCtrl_typ					#
#		· gAxis (to control Slave Moptor)	    as AxisCtrl_typ					#
#																				#
#																				#
#	There are some Libraries needed, too:										#
#		EFILib																	#
#		Libraries (the Global libraries)										#
#																				#
#	And some variables declaration sections:									#
#		GVars: permanent vars are defined in Global.typ., they are needed.		#
#		GStructs: StPermanentGeneral is needed, and it's defined inside it.		#
#																				#
#																				#
#################################################################################
*NOTE: This Package is useless without Analog Thinckness Package to use the outputs of
lasers readings [SEA](30/08/19)

#################################################################################
#################################################################################
#																				#
#			¡¡¡IMPORTANT!!!!													#
# 	Review gAxisCtrl for extra needs about 										#
# 	Axis and Gear to use them													#
#																				#
#################################################################################
```

### Program Logical/ExtPack/_Media/nSensorCtrl/nSensorSim/nSensorSim_v1/nSensorSim (IEC)

#### AllSensors.st
```iecst
ACTION SetAllSensors:
	FOR iIndexSensor:=1 TO data.parameters.iSensorQuantity DO
		data.Inputs.Signals.xPhotoCells[iIndexSensor] := TRUE;
	END_FOR
END_ACTION

ACTION ResetAllSensors:
	FOR iIndexSensor:=1 TO data.parameters.iSensorQuantity DO
		data.Inputs.Signals.xPhotoCells[iIndexSensor] := FALSE;
	END_FOR
END_ACTION
```

#### nSensorSim.st
```iecst
PROGRAM _INIT
	(* Insert code here *)

END_PROGRAM

PROGRAM _CYCLIC
	(* Insert code here *)
	data ACCESS ADR(gPhotoCells);

	rGaugeHeightTillHole := 10.0;

	IF (data.parameters.AlignmentProcess = STP_ALIGNMENT_REQUIRED AND NOT gLine.StatusSummary.xEmptyingBelts) THEN
		//Simulation of the sensors related to the alignement
		IF EDGEPOS(data.status.rPositionMotor > (data.parameters.rSensorMechPositionAlignmentMin - rGaugeHeightTillHole)) THEN
			SetAllSensors;
		ELSIF EDGEPOS(data.status.rPositionMotor > data.parameters.rSensorMechPositionAlignmentMin) THEN
			ResetAllSensors;
		ELSIF EDGEPOS(data.status.rPositionMotor > data.parameters.rSensorMechPositionAlignmentMax) THEN
			SetAllSensors;
		ELSIF EDGEPOS(data.status.rPositionMotor < (data.parameters.rSensorMechPositionAlignmentMin - rGaugeHeightTillHole)) THEN
			ResetAllSensors;
		ELSIF EDGEPOS(ABS(data.status.rPositionMotor-data.status.rSensorPositionAlignment)<0.25) AND data.status.xSensorValidAlignPos THEN
			ResetAllSensors;
		END_IF

		IF 	(data.status.rPositionMotor > data.parameters.rSensorMechPositionMax) OR
			(data.status.rPositionMotor < data.parameters.rSensorMechPositionMin) THEN
			ResetAllSensors;
		END_IF
	END_IF

	IF EDGEPOS(data.commandsSw.xReference) THEN
		ResetAllSensors;
	END_IF

	tonHomingDown.IN := data.status.iSystemState = STP_HOMING_STEP_1;
	tonHomingDown.PT := t#1s;
	tonHomingDown();
	IF tonHomingDown.Q THEN
		data.Inputs.Signals.xPhotoCells[data.parameters.iSensorToReference] := TRUE;
	END_IF

	tonHomingUp.IN := data.status.iSystemState = STP_HOMING_STEP_2;
	tonHomingUp.PT := t#500ms;
	tonHomingUp();
	IF tonHomingUp.Q THEN
		data.Inputs.Signals.xPhotoCells[data.parameters.iSensorToReference] := FALSE;
	END_IF

END_PROGRAM

PROGRAM _EXIT
	(* Insert code here *)

END_PROGRAM
```

### ThicknessAnalog.typ
```iecst
TYPE
	AnalogSensorType :
		(
		ANSENS_BALLUF_48,
		ANSENS_BALLUF_97
		);
	ThicknessAnalogInternal : 	STRUCT
		xMediaToRejectTreated : BOOL; (*Media to Reject has been treated and can be reseted if the sensor is not detecting*)
		xMountedMediaTreated : BOOL; (*Mounted media has been treated and can be reseted if the sensor is not detecting*)
	END_STRUCT;
	stThicknessAnalogAlarms : 	STRUCT
		xMountedTile : BOOL; (*Mlounted Tile Detect*)
		xAlDingDetect : BOOL; (*Stop Alarm*)
		xAlNoDingDetect : BOOL; (*Stop Alarm*)
		xAlDingNotReferenced : BOOL; (*Critical Alarm*)
		xAlDingIncoherenceValue : BOOL; (*Stop Alarm. NOT USING, NOT IN SOFTWARE INTERFACE*)
		xAlDingConexionError : BOOL; (*Stop Alarm*)
		xAlDingNoMediaToCalibrate : BOOL; (*NOT IN ALARM SUMMARY*)
		xAlDingNoDigLaserSensor : BOOL; (*NOT IN ALARM SUMMARY*)
	END_STRUCT;
	stThicknessAnalogIn : 	STRUCT
		pInputCard : UDINT; (*Pointer to the input card of the analog signal*)
		xModuleOK : BOOL; (*PLC card properly connected to X2X*)
		xDingChannelFault : BOOL; (*SoftwareInput*)
		rHighDingMm : REAL; (*AnalogInputCalculate. Value in mm*)
		iHighDingRaw : INT; (*AnalogInput. Direct from the Analog card*)
		xDingHigh : BOOL; (*DI*)
		xDingLow : BOOL; (*DI*)
		xAnyCarriageProductDetect : BOOL; (*Any Product Detect signal coming from Carriage is activated*)
	END_STRUCT;
	stThicknessAnalogOut : 	STRUCT
		xReset : BOOL; (*DO*)
	END_STRUCT;
	stThicknessAnalogState : 	STRUCT
		xDingLowPieceDetect : BOOL; (*DI+Analog value*)
		rCurrentHigh : REAL; (*Current High with offsets. Value in mm*)
		rCurrentThicknessStable : REAL; (*Current High with offsets. Value in mm  Delayed maximum to able to watch it*)
		xDingReferenced : BOOL := FALSE; (*State*)
		xDingInstalled : BOOL; (*State*)
		xSensorCovered : BOOL; (*DI*)
		diLgLowPieceCounter : DINT; (*Log*)
		rOffsetCalibration : REAL; (*Offset to consider the real value of the substrate*)
		rBarsPosition : REAL; (*Minimum position of the bar to avoid a crash. Value in mm*)
		xMediaToRejectDetected : BOOL; (*Media to be rejected has beed detected*)
		xMountedMediaDetected : BOOL; (*Mounted media has been detected*)
		Permanent : stThicknessAnalogPermanent; (*Permanent values stored in flash memory*)
	END_STRUCT;
	stThicknessAnalogPermanent : 	STRUCT
		xDingReferenced : BOOL := FALSE; (*State*)
		rOffsetCalibration : REAL; (*Offset to consider the real value of the substrate*)
	END_STRUCT;
	stThicknessAnalogParametersSw : 	STRUCT
		rCalibrationValue : REAL; (*Software Input. Value of the media in the sensor to adjust the reading*)
	END_STRUCT;
	stThicknessAnalogDiscreteParam : 	STRUCT
		rDistanceBetweenSensors : REAL; (*Distance between the virtual sensors*)
		rOffsetRelToBar : REAL := 0.5; (*Media Offset position in mm. Distance to consider the virtual first digital sensor*)
		iVirtualSensors : USINT; (*Quantity of virtual sensors*)
	END_STRUCT;
	stThicknessAnalogParameters : 	STRUCT
		xDingInstalled : BOOL; (*Configured depending on the machine. Is installed or it can be installed*)
		xEnable : BOOL; (*Configured depending on the machine. Is installed or it can be installed*)
		xAllowDynamicEnable : BOOL; (*The machine allows dynamic enabling or disabling the funcionality*)
		SensorType : AnalogSensorType;
		Discrete : stThicknessAnalogDiscreteParam;
		xKeepHoming : BOOL; (*The system has to keep the homing after a reboot in the PLC*)
		xDiscreteBehavior : BOOL; (*Consider a discrete behavior similar to digital sensors to avoid a lot of movements*)
		xSimulationMode : BOOL; (*Defined by the configuration in Automation Studio*)
		xRaiseDigitalIncoherency : BOOL; (*Raise digital incoherency when receiving Product Detect but not AnalogDetection.Low. Managed in gMachine.Alarms*)
		rMediaThickness : REAL := 5; (*Media Thickness in mm*)
		rMarginPrint : REAL; (*Value in mm*)
		rMachineMinTicknessMedia : REAL; (*Value in mm*)
		MountedDetectionType : ThicknessMountedDetectionType;
		rOverThicknessToMounted : REAL; (*Value in mm over the configured thickness*)
		rThicknessToMounted : REAL; (*Absolute valure in mm to consider mounted*)
		rMountedMediaLevelInBypassMode : REAL; (*mm*)
		rMarginSafePrint : REAL; (*Coming from Sw (indirectly). Fix offset to bent tile. The heads go to the thickness measured + this value. Value in mm*)
		rOverThicknessToReject : REAL; (*mm. Value of the media detected to consider it bad and need to be rejected*)
		rMarginSafeRejectForAnalog : REAL; (*Offset while boards to reject. The heads go to the thickness measured + this value. Value in mm*)
		iAnalogSamples : USINT; (*mm. Value of the media detected to consider it bad and need to be rejected*)
	END_STRUCT;
	stThickessAnalogCommands : 	STRUCT
		xErrorRst : BOOL; (*Order to reset Alarms*)
		xCalibrateThickness : BOOL; (*Software Input*)
		xMute : BOOL; (*Mute Order*)
		AutoMode : stEFI_MachineAutoModes; (*commands to inform belt*)
		Mode : StGeneral_States_Mode;
		xMountedMediaInside : BOOL; (*Mounted Media Inside*)
	END_STRUCT;
	stThicknessAnalog_typ : 	STRUCT
		Alarms : stThicknessAnalogAlarms;
		AlSummary : stEFI_AlarmSummary;
		In : stThicknessAnalogIn;
		Out : stThicknessAnalogOut;
		State : stThicknessAnalogState;
		Parameters : stThicknessAnalogParameters;
		parSw : stThicknessAnalogParametersSw;
		Commands : stThickessAnalogCommands;
		_Internal : nSensorsInternal;
	END_STRUCT;
END_TYPE
```

### Program Logical/ExtPack/_Media/AnalogThicknessCtrl/AnalogThicknessCtrl_v1/Analog_Fast

#### Analog_Fast.st
```iecst
PROGRAM _CYCLIC

	//Access to the Physical inputs
	AnalogInputs;

	///////////////////////
	(*STATES*)
	//////////////////////

	// Getting current high
	gDing.State.rCurrentHigh:= MAX(0, gDing.In.rHighDingMm + gDing.State.rOffsetCalibration);

	// Piece Detect
	gDing.State.xDingLowPieceDetect:= (gDing.State.rCurrentHigh >= gDing.Parameters.rMachineMinTicknessMedia) AND gDing.In.xDingLow;

	xMountedMediaDetected := FALSE;
	xMediaToRejectDetected := FALSE;

	// Alarm: Mounted Tile gui_q_xAlrParoExesoAlturaSet
	// SYSTEM STOPPED DUE TO INPUT SENSORS EXCESSIVE THICKNESS. TO RESET: REMOVE THE TILE FROM THE MACHINE INPUT [12B4]
	IF gDing.Commands.AutoMode.xBypass THEN
		IF gDing.State.xSensorCovered OR gDing.State.rCurrentHigh > gDing.Parameters.rMountedMediaLevelInBypassMode THEN
			xMountedMediaDetected := TRUE;
		END_IF

		IF xMountedMediaDetected AND NOT gDing.Commands.xMountedMediaInside THEN
			gDing.Alarms.xMountedTile:= TRUE;
		END_IF

	ELSIF gDing.Commands.AutoMode.xProdORLab THEN

		// Required to safe printheads installed
		CASE gDing.Parameters.MountedDetectionType OF
			THICKMOUNT_THICKNESS_RELATIVE:
				rThicknessToMounted := gDing.Parameters.rMediaThickness + gDing.Parameters.rOverThicknessToMounted;
			THICKMOUNT_ABSOLUTE:
				rThicknessToMounted := gDing.Parameters.rThicknessToMounted;
		END_CASE

		IF gDing.State.rCurrentHigh > rThicknessToMounted THEN
			xMountedMediaDetected := TRUE;
		END_IF

		// This alarm has to be raised here to avoid resetting it and move out the mounted media
		IF xMountedMediaDetected AND NOT gDing.Commands.xMountedMediaInside THEN
			gDing.Alarms.xMountedTile:= TRUE;
		END_IF

		// MediaToReject
		IF gDing.State.rCurrentHigh > gDing.Parameters.rMediaThickness + gDing.Parameters.rOverThicknessToReject THEN
			xMediaToRejectDetected := TRUE;
		END_IF

	END_IF

	IF xMediaToRejectDetected THEN
		rBarsPosition := gDing.State.rCurrentHigh + gDing.Parameters.rMarginSafeRejectForAnalog;
	ELSE
		IF gDing.Parameters.xDiscreteBehavior THEN
			rBarsPosition := gDing.Parameters.rMediaThickness + gDing.Parameters.rMarginPrint;
			rVirtualDiscretePosition := gDing.Parameters.rMediaThickness + gDing.Parameters.rMarginPrint - gDing.Parameters.Discrete.rOffsetRelToBar;
			FOR iIndexVirtualSensor := 0 TO gDing.Parameters.Discrete.iVirtualSensors -1 DO
				IF gDing.State.rCurrentHigh > rVirtualDiscretePosition + iIndexVirtualSensor * gDing.Parameters.Discrete.rDistanceBetweenSensors - gDing.Parameters.Discrete.rOffsetRelToBar THEN
					rBarsPosition := rVirtualDiscretePosition + ((iIndexVirtualSensor + 1) * gDing.Parameters.Discrete.rDistanceBetweenSensors );
				END_IF
			END_FOR
		ELSE
			rBarsPosition := gDing.State.rCurrentHigh + gDing._Internal.rMarginSafePrintChecked;
		END_IF
	END_IF

	gDing.State.rBarsPosition := rBarsPosition;

	// Data has to be treated in the slow program to be sure to read the information in all fast programs
	IF xMountedMediaDetected (*AND NOT gDing._Internal.xMountedMediaTreated*) THEN
		gDing.State.xMountedMediaDetected := TRUE;
	ELSIF NOT xMountedMediaDetected AND gDing._Internal.xMountedMediaTreated THEN
		gDing.State.xMountedMediaDetected := FALSE;
	END_IF

	// Data has to be treated in the slow program to be sure to read the information in all fast programs
	IF xMediaToRejectDetected (*AND NOT gDing._Internal.xMediaToRejectTreated*) THEN
		gDing.State.xMediaToRejectDetected := TRUE;
	ELSIF NOT xMediaToRejectDetected AND gDing._Internal.xMediaToRejectTreated THEN
		gDing.State.xMediaToRejectDetected := FALSE;
	END_IF

END_PROGRAM
```

#### AnalogInputs.st
```iecst
ACTION AnalogInputs:

	//If in simulation, do not assign physical mapping
	IF gDing.Parameters.xSimulationMode THEN
		RETURN;
	END_IF

	//If not installed, clear alarms and exit
	IF NOT gDing.Parameters.xDingInstalled THEN
		gDing.State.xDingLowPieceDetect := FALSE;
		RETURN;
	END_IF

	// If the pointer of the card is not assigned by machine,
	//return to avoid lost pointer access
	IF gDing.In.pInputCard = 0 THEN
		RETURN;
	END_IF

	dingCard ACCESS gDing.In.pInputCard;

	// Analog Input
	IF dingCard.AInput[1] < 5 OR gDing.In.xDingChannelFault THEN
		gDing.In.iHighDingRaw:=0;
		gDing.In.rHighDingMm:=0;
	ELSIF dingCard.AInput[1] > 6543 THEN // Rename Analog Input
		//Taking the maximum because the AnalogInputCard

		// Calculating and checking MaxSamples
		iMaxSamples := MIN(MAX_LAST_SIGNAL, gDing.Parameters.iAnalogSamples);

		// Calculating the Max from the samples
		iHighDingRaw := dingCard.AInput[1];
		FOR iIndexSamples := 2 TO iMaxSamples DO
			iHighDingRaw := MAX(iHighDingRaw, dingCard.AInput[iIndexSamples]);
		END_FOR
		gDing.In.iHighDingRaw := iHighDingRaw;

		gDing.State.xSensorCovered:= gDing.In.iHighDingRaw > 32700;

		CASE gDing.Parameters.SensorType OF
			ANSENS_BALLUF_48:
				gDing.In.rHighDingMm:=INT_TO_REAL(gDing.In.iHighDingRaw - 6543) * ((48.76 / (32767.0- 6543.0))  );

			ANSENS_BALLUF_97:
				gDing.In.rHighDingMm:=INT_TO_REAL(gDing.In.iHighDingRaw - 6543) * ((97.53 / (32767.0- 6543.0))  );

		END_CASE

	END_IF

END_ACTION
```

### Program Logical/ExtPack/_Media/AnalogThicknessCtrl/AnalogThicknessCtrl_v1/AnalogThickness (IEC)

#### Reset.st
```iecst
ACTION ResetAlarms:
	data.Alarms := stThickAlarmsReseted;
	data.AlSummary := stAlarmsSummaryReseted;
END_ACTION

ACTION ResetCommands:
	data.Commands:=CommandsReseted;
END_ACTION
```

#### AlarmsSummary.st - Alarms summary
```iecst
ACTION AlarmsSummary:

	//////////////////////////
	////// RESET ALARMS //////
	//////////////////////////
	// Pending do commands gdata.commands.xReset
	IF data.Commands.xErrorRst THEN
		data.Alarms := stThickAlarmsReseted;
		data.AlSummary := stAlarmsSummaryReseted;
	END_IF

	//Alarms STOP
	iReasonStop.0 := data.Alarms.xAlDingConexionError;
	iReasonStop.1 := data.Alarms.xAlDingNotReferenced;
	iReasonStop.2 := data.Alarms.xAlDingDetect;
	iReasonStop.3 := data.Alarms.xAlNoDingDetect;
	iReasonStop.4 := data.Alarms.xAlDingIncoherenceValue;
	iReasonStop.5 := data.Alarms.xAlDingNoDigLaserSensor;

	data.AlSummary.xAlarmStop := iReasonStop > 0;
	IF EDGEPOS(data.AlSummary.xAlarmStop) THEN
		data.AlSummary.iReasonStop[0] := iReasonStop;
	ELSIF EDGEPOS(NOT data.Commands.AutoMode.xStop AND NOT data.AlSummary.xAlarmStop) THEN
		data.AlSummary.iReasonStop[0] := 0;
	END_IF

	//Alarms CRITICAL
	iReasonCritical.0 := data.Alarms.xAlDingConexionError AND data.Commands.AutoMode.xProdORLab;

	data.AlSummary.xAlarmCritical := iReasonCritical > 0;
	IF data.Commands.Mode.xAuto AND EDGEPOS(data.AlSummary.xAlarmCritical) THEN
		data.AlSummary.iReasonCritical := iReasonCritical;
	ELSIF EDGEPOS(data.Commands.Mode.xAuto AND NOT data.AlSummary.xAlarmCritical) THEN
		data.AlSummary.iReasonCritical := 0;
	END_IF

END_ACTION
```

#### AnalogThickness.var - Local variables
```iecst
VAR CONSTANT
	VALUES_TO_GET_MAX_THICKNESS : USINT := 99;
END_VAR
VAR
	T_NoDigDingDetect : TON;
	stAlarmsSummaryReseted : stEFI_AlarmSummary;
	stThickAlarmsReseted : stThicknessAnalogAlarms;
	stEventLogCal : EventLog_typ;
	stEventLog : EventLog_typ;
	stEventLogReject : EventLog_typ;
	stEventLogEndReject : EventLog_typ;
	strAux : STRING[129];
	iReasonStop : UDINT;
	iReasonCritical : UDINT;
	CommandsReseted : stThickessAnalogCommands;
	rMaxThicknessS1 : REAL;
	rMaxThicknessS2 : REAL;
	rMaxThicknessS0 : REAL;
	rMaxThickness : REAL;
	iModSec : USINT;
	timeReaded : RTCtime_typ;
	ars_AlDingConexionError : AutoResetSound;
	ars_AlDingNotReferenced : AutoResetSound;
	ars_AlDingDetect : AutoResetSound;
	ars_AlNoDingDetect : AutoResetSound;
	ars_AlDingIncoherenceValue : AutoResetSound;
	ars_AlDingNoDigLaserSensor : AutoResetSound;
	ars_AlMountedTile : AutoResetSound;
	data : REFERENCE TO stThicknessAnalog_typ;
	xRecoveredPermanentInfo : BOOL;
END_VAR
```

### BasicDetectMediaCtrl.typ
```iecst
TYPE
	DetectionMedia_Parameters : 	STRUCT
		xInstalled : BOOL;
		xBeltMoving : BOOL; (*The belt is moving*)
		rCorrection : REAL;
		rDesiredHeigh : REAL; (*Value in mm*)
	END_STRUCT;
	DetectionMedia_Inputs : 	STRUCT
		xMountedMedia : BOOL;
		xMediaPresentL1 : BOOL;
		xMediaPresentL2 : BOOL;
		xCorrection : BOOL;
	END_STRUCT;
	DetectionMedia_Alarms : 	STRUCT
		xMountedMedia : BOOL;
	END_STRUCT;
	DetectionMedia_Status : 	STRUCT
		xInstalled : BOOL;
		xMediaPresent : BOOL;
		rMediaHeigh : REAL; (*Value in mm*)
	END_STRUCT;
	DetectionMedia_Commands : 	STRUCT
		xReset : BOOL; (*Order to reset Alarms*)
		xMute : BOOL; (*Mute Order*)
		StateMode : enumEFI_GenMachineState; (*commands to inform belt*)
		AutoMode : stEFI_MachineAutoModes; (*commands to inform belt*)
	END_STRUCT;
	DetectionMedia : 	STRUCT
		Inputs : DetectionMedia_Inputs;
		Parameters : DetectionMedia_Parameters;
		Commands : DetectionMedia_Commands;
		Status : DetectionMedia_Status;
		Alarms : DetectionMedia_Alarms;
		AlSummary : stEFI_AlarmSummary;
	END_STRUCT;
END_TYPE
```

### Program Logical/ExtPack/_Motion/AxisCtrl/AxisCtrl_v2/AxisCtrl (IEC, version 0.02.7) - Axis logical control
